PROGRAM Gate_Big_Move
VAR
	bigGateGearIn			:MC_GearInDyn;			// 大龙门电子齿轮，LeftAxis为Master
	bigGateLeftAxisJog		:MC_Jog;				// 大龙门左轴(电子齿轮的Master轴)MC_Jog
END_VAR

bigGateGearIn(
	Master:= axis_BigGate_Left, 
	Slave:= axis_BigGate_Right, 
	Enable:= TRUE, 
	GearRatio:= -1.0, 
	Acceleration:= , 
	Deceleration:= , 
	Jerk:= , 
	BufferMode:= , 
	Options:= , 
	InGear=> , 
	Busy=> , 
	Active=> , 
	CommandAborted=> , 
	Error=> , 
	ErrorID=> );

	
bigGateLeftAxisJog(
	Axis:= axis_BigGate_Left, 
	JogForward:= bBigGate_Up, 
	JogBackwards:= bBigGate_Down, 
	Mode:= , 
	Position:= , 
	Velocity:= , 
	Acceleration:= , 
	Deceleration:= , 
	Jerk:= , 
	Done=> , 
	Busy=> , 
	Active=> , 
	CommandAborted=> , 
	Error=> , 
	ErrorID=> );

END_PROGRAM

(* stored: Version 1.1.0.1, ProductVersion 3.1.4024.14
   POU Gate_Big_Move: Id {d13f1184-948a-47c6-a403-9da76bad7ac5}, SpecialFunc None *)
